// TIA Portal V20 export
FUNCTION_BLOCK "FB2002_Axis_Function"   // FB2, LAD
{ S7_Optimized_Access := 'TRUE' }
// stored: MemoryReserve 100, SetENOAutomatically false
   VAR_INPUT
      Plant_Identifier { ExternalAccessible := 'False'; ExternalVisible := 'False'; ExternalWritable := 'False'} : WString[24];
      Opmode { ExternalAccessible := 'False'; ExternalVisible := 'False'; ExternalWritable := 'False'} : "OPMODE_OUT_UDT";
      TO_Pos_Axis : TO_PositioningAxis;
      Axis_Nr : Int;
      Axis_AbsNum : Int;
      I_SS_bHome : Bool;   // 原点传感器
      I_SS_bFW : Bool := TRUE;   // 前限位
      I_SS_bBW : Bool := TRUE;   // 后限位
      I_CMD_bEnableAxis : Bool;   // 使能
      I_CMD_bResetAxis : Bool;   // 复位
      I_CMD_bjogForward : Bool;   // Taster Aufwärts / 正点
      I_CMD_bjogBackward : Bool;   // Taster Abwärts / 反点
      I_CMD_bmoveVelocity : Bool;   // 速度运行
      I_CMD_bstop : Bool;   // 停止
      I_CMD_bfastStop : Bool;   // 急停
      I_CMD_bHoming : Bool;   // 回零
      I_CMD_bGoToPos : Array[0..15] of Bool;   // Start Aufwärts in Automatik / 16个定位
      I_CMD_iGoToPos : Word;   // 16个定位 Word
      I_CMD_bCallAbsPos : Bool;   // 定位位置切换时，单独的定位按钮
      I_CMD_bRelPos : Bool;   // 相对定位
      I_InLock_bEnableAxis : Bool;   // 使能
      I_InLock_bResetAxis : Bool;   // 复位
      I_InLock_bjogForward : Bool;   // Taster Aufwärts / 正点
      I_InLock_bjogBackward : Bool;   // Taster Abwärts / 反点
      I_InLock_bmoveVelocity : Bool;   // 速度运行
      I_InLock_bstop : Bool;   // 停止
      I_InLock_bfastStop : Bool;   // 急停
      I_InLock_bHoming : Bool;   // 回零
      I_InLock_bGoToPos : Array[0..16] of Bool;   // Start Aufwärts in Automatik / 16个定位
      I_InLock_iGoToPos : Word;   // 16个定位 Word
      I_InLock_bCallAbsPos : Bool;   // 定位位置切换时，单独的定位按钮
      I_InLock_bRelPos : Bool;   // 相对定位
      I_InLock_MyBool : Array[0..5] of Bool;   // 临时变量
      I_CMD_bGoToPos_0 : Bool;   // Start Aufwärts in Automatik / 16个定位自动
      I_InLock_bGoToPos_0 : Bool;   // Start Aufwärts in Automatik / 16个定位条件
      I_CMD_bGoToPos_1 : Bool;   // Start Aufwärts in Automatik / 16个定位自动
      I_InLock_bGoToPos_1 : Bool;   // Start Aufwärts in Automatik / 16个定位条件
      I_CMD_bGoToPos_2 : Bool;   // Start Aufwärts in Automatik / 16个定位自动
      I_InLock_bGoToPos_2 : Bool;   // Start Aufwärts in Automatik / 16个定位条件
      I_CMD_bGoToPos_3 : Bool;   // Start Aufwärts in Automatik / 16个定位自动
      I_InLock_bGoToPos_3 : Bool;   // Start Aufwärts in Automatik / 16个定位条件
      I_CMD_bGoToPos_4 : Bool;   // Start Aufwärts in Automatik / 16个定位自动
      I_InLock_bGoToPos_4 : Bool;   // Start Aufwärts in Automatik / 16个定位条件
      I_CMD_bGoToPos_5 : Bool;   // Start Aufwärts in Automatik / 16个定位自动
      I_InLock_bGoToPos_5 : Bool;   // Start Aufwärts in Automatik / 16个定位条件
      I_CMD_bGoToPos_6 : Bool;   // Start Aufwärts in Automatik / 16个定位自动
      I_InLock_bGoToPos_6 : Bool;   // Start Aufwärts in Automatik / 16个定位条件
      I_CMD_bGoToPos_7 : Bool;   // Start Aufwärts in Automatik / 16个定位自动
      I_InLock_bGoToPos_7 : Bool;   // Start Aufwärts in Automatik / 16个定位条件
      I_CMD_bGoToPos_8 : Bool;   // Start Aufwärts in Automatik / 16个定位自动
      I_InLock_bGoToPos_8 : Bool;   // Start Aufwärts in Automatik / 16个定位条件
   END_VAR
   VAR_OUTPUT
      O_Status_bAxisReady : Bool;   // 轴通讯正常
      O_Status_bAxisEnabled : Bool;   // 轴使能
      O_Status_bjogForward : Bool;   // 轴正点中
      O_Status_bjogBackward : Bool;   // 轴反点中
      O_Status_bHomed : Bool;   // 轴归零完成
      O_Status_bAtHome : Bool;   // 轴在零位
      O_Status_bSstill : Bool;   // 轴静止
      O_Status_bAxisBusy : Bool;   // 轴运行中
      O_Status_bAxisSyned : Bool;   // 同步上
      O_Status_bAxisError : Bool;   // 轴报警
      O_Status_bAtPos : Array[0..15] of Bool;   // Ausgang Aufwärts / 在目标位置上
      O_Status_bPosDone : Array[0..15] of Bool;   // 定位完成
      O_Status_bPosing : Array[0..15] of Bool;   // Ausgang Aufwärts / 定位中
      O_Status_bRelPosDone : Bool;   // 相对定位完成
      O_Status_rActPos : LReal;   // 实际位置
      O_Status_rActSpeed : LReal;   // 实际速度
      O_Status_iAxisFaultNum : UDInt;   // 轴报警代码
      O_Status_iDriveFaultNum : UDInt;   // 驱动报警代码
      O_Status_iFBStatus : Word;   // 运动功能块状态
      O_Status_iMCStatus : Word;   // 运动指令状态
      O_Status_rDriveTorque : LReal;   // 驱动扭矩
      O_Status_rDriveTemp : LReal;   // 驱动温度
      O_Status_rDriveRpm : LReal;   // 驱动转速
      O_Status_AxisName : WString[24] := WSTRING#'No axis';   // Name of axis
      O_Status_mybool : Array[0..5] of Bool;   // 备用
      O_Status_myLreal : Array[0..5] of LReal;   // 备用
   END_VAR
   VAR_IN_OUT
      IF_HMI : "Axis_IF_HMI";
   END_VAR
   VAR
      myFB_Pos16_Ax01 { S7_SetPoint := 'True'} : "FB_Pos16_IO";
      Axis_01 { S7_SetPoint := 'True'} : "FB_Axis";
      i { ExternalAccessible := 'False'; ExternalVisible := 'False'; ExternalWritable := 'False'} : Int;
      j { ExternalAccessible := 'False'; ExternalVisible := 'False'; ExternalWritable := 'False'} : Int;
      HOMIEDONE : Bool;
   END_VAR
BEGIN

REGION Network 1
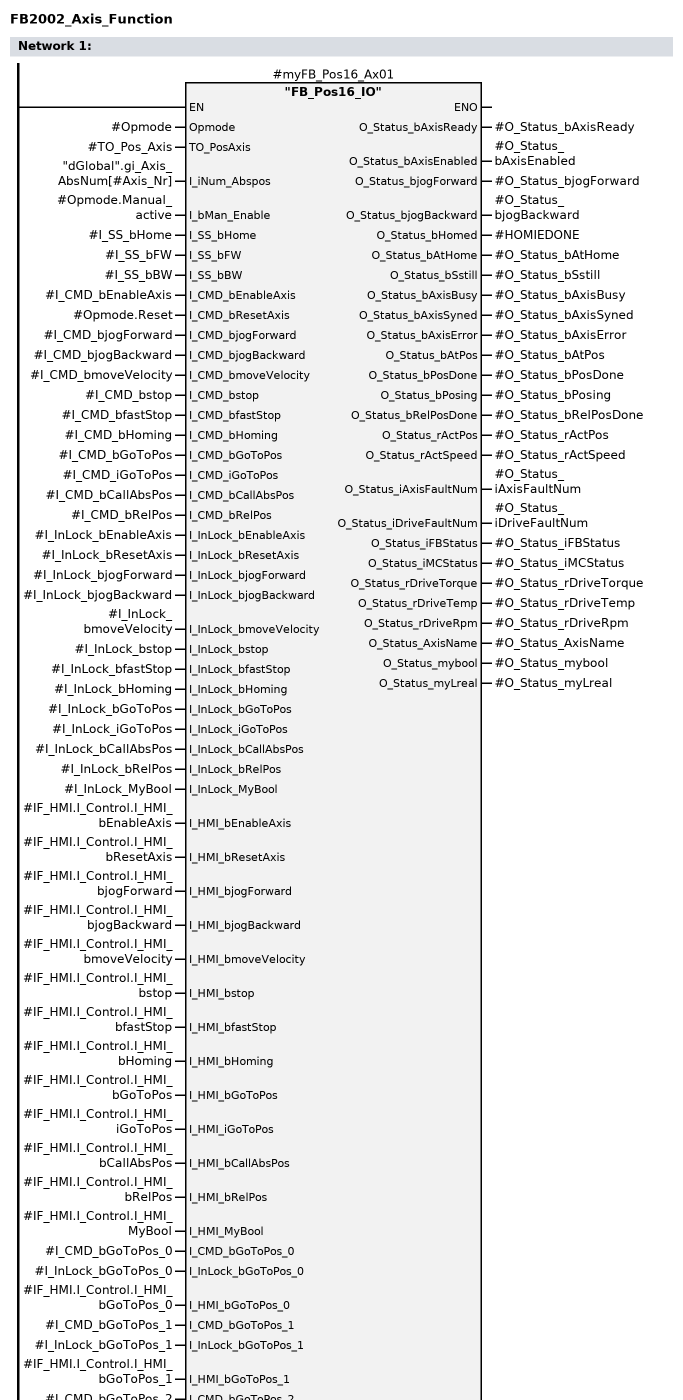
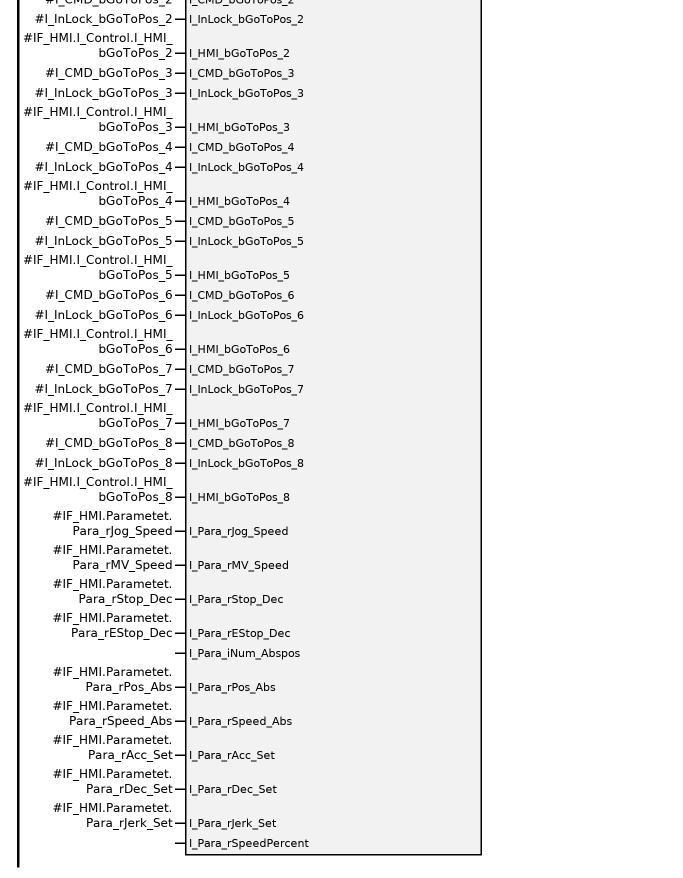
   RUNG wire#powerrail
      #myFB_Pos16_Ax01(Opmode := #Opmode, TO_PosAxis := #TO_Pos_Axis, I_iNum_Abspos := "dGlobal".gi_Axis_AbsNum[#Axis_Nr], I_bMan_Enable := #Opmode.Manual_active, I_SS_bHome := #I_SS_bHome, I_SS_bFW := #I_SS_bFW, I_SS_bBW := #I_SS_bBW, I_CMD_bEnableAxis := #I_CMD_bEnableAxis, I_CMD_bResetAxis := #Opmode.Reset, I_CMD_bjogForward := #I_CMD_bjogForward, I_CMD_bjogBackward := #I_CMD_bjogBackward, I_CMD_bmoveVelocity := #I_CMD_bmoveVelocity, I_CMD_bstop := #I_CMD_bstop, I_CMD_bfastStop := #I_CMD_bfastStop, I_CMD_bHoming := #I_CMD_bHoming, I_CMD_bGoToPos := #I_CMD_bGoToPos, I_CMD_iGoToPos := #I_CMD_iGoToPos, I_CMD_bCallAbsPos := #I_CMD_bCallAbsPos, I_CMD_bRelPos := #I_CMD_bRelPos, I_InLock_bEnableAxis := #I_InLock_bEnableAxis, I_InLock_bResetAxis := #I_InLock_bResetAxis, I_InLock_bjogForward := #I_InLock_bjogForward, I_InLock_bjogBackward := #I_InLock_bjogBackward, I_InLock_bmoveVelocity := #I_InLock_bmoveVelocity, I_InLock_bstop := #I_InLock_bstop, I_InLock_bfastStop := #I_InLock_bfastStop, I_InLock_bHoming := #I_InLock_bHoming, I_InLock_bGoToPos := #I_InLock_bGoToPos, I_InLock_iGoToPos := #I_InLock_iGoToPos, I_InLock_bCallAbsPos := #I_InLock_bCallAbsPos, I_InLock_bRelPos := #I_InLock_bRelPos, I_InLock_MyBool := #I_InLock_MyBool, I_HMI_bEnableAxis := #IF_HMI.I_Control.I_HMI_bEnableAxis, I_HMI_bResetAxis := #IF_HMI.I_Control.I_HMI_bResetAxis, I_HMI_bjogForward := #IF_HMI.I_Control.I_HMI_bjogForward, I_HMI_bjogBackward := #IF_HMI.I_Control.I_HMI_bjogBackward, I_HMI_bmoveVelocity := #IF_HMI.I_Control.I_HMI_bmoveVelocity, I_HMI_bstop := #IF_HMI.I_Control.I_HMI_bstop, I_HMI_bfastStop := #IF_HMI.I_Control.I_HMI_bfastStop, I_HMI_bHoming := #IF_HMI.I_Control.I_HMI_bHoming, I_HMI_bGoToPos := #IF_HMI.I_Control.I_HMI_bGoToPos, I_HMI_iGoToPos := #IF_HMI.I_Control.I_HMI_iGoToPos, I_HMI_bCallAbsPos := #IF_HMI.I_Control.I_HMI_bCallAbsPos, I_HMI_bRelPos := #IF_HMI.I_Control.I_HMI_bRelPos, I_HMI_MyBool := #IF_HMI.I_Control.I_HMI_MyBool, I_CMD_bGoToPos_0 := #I_CMD_bGoToPos_0, I_InLock_bGoToPos_0 := #I_InLock_bGoToPos_0, I_HMI_bGoToPos_0 := #IF_HMI.I_Control.I_HMI_bGoToPos_0, I_CMD_bGoToPos_1 := #I_CMD_bGoToPos_1, I_InLock_bGoToPos_1 := #I_InLock_bGoToPos_1, I_HMI_bGoToPos_1 := #IF_HMI.I_Control.I_HMI_bGoToPos_1, I_CMD_bGoToPos_2 := #I_CMD_bGoToPos_2, I_InLock_bGoToPos_2 := #I_InLock_bGoToPos_2, I_HMI_bGoToPos_2 := #IF_HMI.I_Control.I_HMI_bGoToPos_2, I_CMD_bGoToPos_3 := #I_CMD_bGoToPos_3, I_InLock_bGoToPos_3 := #I_InLock_bGoToPos_3, I_HMI_bGoToPos_3 := #IF_HMI.I_Control.I_HMI_bGoToPos_3, I_CMD_bGoToPos_4 := #I_CMD_bGoToPos_4, I_InLock_bGoToPos_4 := #I_InLock_bGoToPos_4, I_HMI_bGoToPos_4 := #IF_HMI.I_Control.I_HMI_bGoToPos_4, I_CMD_bGoToPos_5 := #I_CMD_bGoToPos_5, I_InLock_bGoToPos_5 := #I_InLock_bGoToPos_5, I_HMI_bGoToPos_5 := #IF_HMI.I_Control.I_HMI_bGoToPos_5, I_CMD_bGoToPos_6 := #I_CMD_bGoToPos_6, I_InLock_bGoToPos_6 := #I_InLock_bGoToPos_6, I_HMI_bGoToPos_6 := #IF_HMI.I_Control.I_HMI_bGoToPos_6, I_CMD_bGoToPos_7 := #I_CMD_bGoToPos_7, I_InLock_bGoToPos_7 := #I_InLock_bGoToPos_7, I_HMI_bGoToPos_7 := #IF_HMI.I_Control.I_HMI_bGoToPos_7, I_CMD_bGoToPos_8 := #I_CMD_bGoToPos_8, I_InLock_bGoToPos_8 := #I_InLock_bGoToPos_8, I_HMI_bGoToPos_8 := #IF_HMI.I_Control.I_HMI_bGoToPos_8, I_Para_rJog_Speed := #IF_HMI.Parametet.Para_rJog_Speed, I_Para_rMV_Speed := #IF_HMI.Parametet.Para_rMV_Speed, I_Para_rStop_Dec := #IF_HMI.Parametet.Para_rStop_Dec, I_Para_rEStop_Dec := #IF_HMI.Parametet.Para_rEStop_Dec, I_Para_iNum_Abspos :=, I_Para_rPos_Abs := #IF_HMI.Parametet.Para_rPos_Abs, I_Para_rSpeed_Abs := #IF_HMI.Parametet.Para_rSpeed_Abs, I_Para_rAcc_Set := #IF_HMI.Parametet.Para_rAcc_Set, I_Para_rDec_Set := #IF_HMI.Parametet.Para_rDec_Set, I_Para_rJerk_Set := #IF_HMI.Parametet.Para_rJerk_Set, I_Para_rSpeedPercent :=, O_Status_bAxisReady => #O_Status_bAxisReady, O_Status_bAxisEnabled => #O_Status_bAxisEnabled, O_Status_bjogForward => #O_Status_bjogForward, O_Status_bjogBackward => #O_Status_bjogBackward, O_Status_bHomed => #HOMIEDONE, O_Status_bAtHome => #O_Status_bAtHome, O_Status_bSstill => #O_Status_bSstill, O_Status_bAxisBusy => #O_Status_bAxisBusy, O_Status_bAxisSyned => #O_Status_bAxisSyned, O_Status_bAxisError => #O_Status_bAxisError, O_Status_bAtPos => #O_Status_bAtPos, O_Status_bPosDone => #O_Status_bPosDone, O_Status_bPosing => #O_Status_bPosing, O_Status_bRelPosDone => #O_Status_bRelPosDone, O_Status_rActPos => #O_Status_rActPos, O_Status_rActSpeed => #O_Status_rActSpeed, O_Status_iAxisFaultNum => #O_Status_iAxisFaultNum, O_Status_iDriveFaultNum => #O_Status_iDriveFaultNum, O_Status_iFBStatus => #O_Status_iFBStatus, O_Status_iMCStatus => #O_Status_iMCStatus, O_Status_rDriveTorque => #O_Status_rDriveTorque, O_Status_rDriveTemp => #O_Status_rDriveTemp, O_Status_rDriveRpm => #O_Status_rDriveRpm, O_Status_AxisName => #O_Status_AxisName, O_Status_mybool => #O_Status_mybool, O_Status_myLreal => #O_Status_myLreal)
   END_RUNG
   // the same network as SCL:
   #myFB_Pos16_Ax01(Opmode := #Opmode,   // "FB_Pos16_IO"
                    TO_PosAxis := #TO_Pos_Axis,
                    I_iNum_Abspos := "dGlobal".gi_Axis_AbsNum[#Axis_Nr],
                    I_bMan_Enable := #Opmode.Manual_active,
                    I_SS_bHome := #I_SS_bHome,
                    I_SS_bFW := #I_SS_bFW,
                    I_SS_bBW := #I_SS_bBW,
                    I_CMD_bEnableAxis := #I_CMD_bEnableAxis,
                    I_CMD_bResetAxis := #Opmode.Reset,
                    I_CMD_bjogForward := #I_CMD_bjogForward,
                    I_CMD_bjogBackward := #I_CMD_bjogBackward,
                    I_CMD_bmoveVelocity := #I_CMD_bmoveVelocity,
                    I_CMD_bstop := #I_CMD_bstop,
                    I_CMD_bfastStop := #I_CMD_bfastStop,
                    I_CMD_bHoming := #I_CMD_bHoming,
                    I_CMD_bGoToPos := #I_CMD_bGoToPos,
                    I_CMD_iGoToPos := #I_CMD_iGoToPos,
                    I_CMD_bCallAbsPos := #I_CMD_bCallAbsPos,
                    I_CMD_bRelPos := #I_CMD_bRelPos,
                    I_InLock_bEnableAxis := #I_InLock_bEnableAxis,
                    I_InLock_bResetAxis := #I_InLock_bResetAxis,
                    I_InLock_bjogForward := #I_InLock_bjogForward,
                    I_InLock_bjogBackward := #I_InLock_bjogBackward,
                    I_InLock_bmoveVelocity := #I_InLock_bmoveVelocity,
                    I_InLock_bstop := #I_InLock_bstop,
                    I_InLock_bfastStop := #I_InLock_bfastStop,
                    I_InLock_bHoming := #I_InLock_bHoming,
                    I_InLock_bGoToPos := #I_InLock_bGoToPos,
                    I_InLock_iGoToPos := #I_InLock_iGoToPos,
                    I_InLock_bCallAbsPos := #I_InLock_bCallAbsPos,
                    I_InLock_bRelPos := #I_InLock_bRelPos,
                    I_InLock_MyBool := #I_InLock_MyBool,
                    I_HMI_bEnableAxis := #IF_HMI.I_Control.I_HMI_bEnableAxis,
                    I_HMI_bResetAxis := #IF_HMI.I_Control.I_HMI_bResetAxis,
                    I_HMI_bjogForward := #IF_HMI.I_Control.I_HMI_bjogForward,
                    I_HMI_bjogBackward := #IF_HMI.I_Control.I_HMI_bjogBackward,
                    I_HMI_bmoveVelocity := #IF_HMI.I_Control.I_HMI_bmoveVelocity,
                    I_HMI_bstop := #IF_HMI.I_Control.I_HMI_bstop,
                    I_HMI_bfastStop := #IF_HMI.I_Control.I_HMI_bfastStop,
                    I_HMI_bHoming := #IF_HMI.I_Control.I_HMI_bHoming,
                    I_HMI_bGoToPos := #IF_HMI.I_Control.I_HMI_bGoToPos,
                    I_HMI_iGoToPos := #IF_HMI.I_Control.I_HMI_iGoToPos,
                    I_HMI_bCallAbsPos := #IF_HMI.I_Control.I_HMI_bCallAbsPos,
                    I_HMI_bRelPos := #IF_HMI.I_Control.I_HMI_bRelPos,
                    I_HMI_MyBool := #IF_HMI.I_Control.I_HMI_MyBool,
                    I_CMD_bGoToPos_0 := #I_CMD_bGoToPos_0,
                    I_InLock_bGoToPos_0 := #I_InLock_bGoToPos_0,
                    I_HMI_bGoToPos_0 := #IF_HMI.I_Control.I_HMI_bGoToPos_0,
                    I_CMD_bGoToPos_1 := #I_CMD_bGoToPos_1,
                    I_InLock_bGoToPos_1 := #I_InLock_bGoToPos_1,
                    I_HMI_bGoToPos_1 := #IF_HMI.I_Control.I_HMI_bGoToPos_1,
                    I_CMD_bGoToPos_2 := #I_CMD_bGoToPos_2,
                    I_InLock_bGoToPos_2 := #I_InLock_bGoToPos_2,
                    I_HMI_bGoToPos_2 := #IF_HMI.I_Control.I_HMI_bGoToPos_2,
                    I_CMD_bGoToPos_3 := #I_CMD_bGoToPos_3,
                    I_InLock_bGoToPos_3 := #I_InLock_bGoToPos_3,
                    I_HMI_bGoToPos_3 := #IF_HMI.I_Control.I_HMI_bGoToPos_3,
                    I_CMD_bGoToPos_4 := #I_CMD_bGoToPos_4,
                    I_InLock_bGoToPos_4 := #I_InLock_bGoToPos_4,
                    I_HMI_bGoToPos_4 := #IF_HMI.I_Control.I_HMI_bGoToPos_4,
                    I_CMD_bGoToPos_5 := #I_CMD_bGoToPos_5,
                    I_InLock_bGoToPos_5 := #I_InLock_bGoToPos_5,
                    I_HMI_bGoToPos_5 := #IF_HMI.I_Control.I_HMI_bGoToPos_5,
                    I_CMD_bGoToPos_6 := #I_CMD_bGoToPos_6,
                    I_InLock_bGoToPos_6 := #I_InLock_bGoToPos_6,
                    I_HMI_bGoToPos_6 := #IF_HMI.I_Control.I_HMI_bGoToPos_6,
                    I_CMD_bGoToPos_7 := #I_CMD_bGoToPos_7,
                    I_InLock_bGoToPos_7 := #I_InLock_bGoToPos_7,
                    I_HMI_bGoToPos_7 := #IF_HMI.I_Control.I_HMI_bGoToPos_7,
                    I_CMD_bGoToPos_8 := #I_CMD_bGoToPos_8,
                    I_InLock_bGoToPos_8 := #I_InLock_bGoToPos_8,
                    I_HMI_bGoToPos_8 := #IF_HMI.I_Control.I_HMI_bGoToPos_8,
                    I_Para_rJog_Speed := #IF_HMI.Parametet.Para_rJog_Speed,
                    I_Para_rMV_Speed := #IF_HMI.Parametet.Para_rMV_Speed,
                    I_Para_rStop_Dec := #IF_HMI.Parametet.Para_rStop_Dec,
                    I_Para_rEStop_Dec := #IF_HMI.Parametet.Para_rEStop_Dec,
                    I_Para_rPos_Abs := #IF_HMI.Parametet.Para_rPos_Abs,
                    I_Para_rSpeed_Abs := #IF_HMI.Parametet.Para_rSpeed_Abs,
                    I_Para_rAcc_Set := #IF_HMI.Parametet.Para_rAcc_Set,
                    I_Para_rDec_Set := #IF_HMI.Parametet.Para_rDec_Set,
                    I_Para_rJerk_Set := #IF_HMI.Parametet.Para_rJerk_Set,
                    O_Status_bAxisReady => #O_Status_bAxisReady,
                    O_Status_bAxisEnabled => #O_Status_bAxisEnabled,
                    O_Status_bjogForward => #O_Status_bjogForward,
                    O_Status_bjogBackward => #O_Status_bjogBackward,
                    O_Status_bHomed => #HOMIEDONE,
                    O_Status_bAtHome => #O_Status_bAtHome,
                    O_Status_bSstill => #O_Status_bSstill,
                    O_Status_bAxisBusy => #O_Status_bAxisBusy,
                    O_Status_bAxisSyned => #O_Status_bAxisSyned,
                    O_Status_bAxisError => #O_Status_bAxisError,
                    O_Status_bAtPos => #O_Status_bAtPos,
                    O_Status_bPosDone => #O_Status_bPosDone,
                    O_Status_bPosing => #O_Status_bPosing,
                    O_Status_bRelPosDone => #O_Status_bRelPosDone,
                    O_Status_rActPos => #O_Status_rActPos,
                    O_Status_rActSpeed => #O_Status_rActSpeed,
                    O_Status_iAxisFaultNum => #O_Status_iAxisFaultNum,
                    O_Status_iDriveFaultNum => #O_Status_iDriveFaultNum,
                    O_Status_iFBStatus => #O_Status_iFBStatus,
                    O_Status_iMCStatus => #O_Status_iMCStatus,
                    O_Status_rDriveTorque => #O_Status_rDriveTorque,
                    O_Status_rDriveTemp => #O_Status_rDriveTemp,
                    O_Status_rDriveRpm => #O_Status_rDriveRpm,
                    O_Status_AxisName => #O_Status_AxisName,
                    O_Status_mybool => #O_Status_mybool,
                    O_Status_myLreal => #O_Status_myLreal);
END_REGION

REGION Network 2 (SCL)
   IF #HOMIEDONE THEN
       #O_Status_bHomed := 1;
   END_IF;
   IF #O_Status_rActSpeed>0.5 THEN
           #O_Status_bHomed := 0;
   END_IF;
END_REGION

REGION Network 4 (SCL)


       "dGlobal".gi_Axis_AbsNum[#Axis_Nr] := #Axis_AbsNum;
END_REGION

REGION Network 6 (SCL)

       "dStruct_Axis".gs_Axis[#Axis_Nr].I_CMD.bResetAxis := #Opmode.Reset;
       "dStruct_Axis".gs_Axis[#Axis_Nr].I_InLock.bjogForward := "dStruct_Axis".gs_Axis[#Axis_Nr].O_Status.bAxisEnabled;
       "dStruct_Axis".gs_Axis[#Axis_Nr].I_InLock.bjogBackward := "dStruct_Axis".gs_Axis[#Axis_Nr].O_Status.bAxisEnabled;
       "dStruct_Axis".gs_Axis[#Axis_Nr].I_InLock.bHoming := true;
       FOR #j := 0 TO 16 DO
           "dStruct_Axis".gs_Axis[#Axis_Nr].I_InLock.bGoToPos[#j] := true;
       END_FOR;


       IF "dGlobal".Old_Pos_Select <> "dGlobal".gbo_Pos_Select THEN//刚切换
           "dStruct_Axis".gs_Axis[0].I_Para.rPos_Abs[0] := "dStruct_Axis".gs_Axis["dGlobal".gbo_Axis_Select].I_Para.rPos_Abs["dGlobal".gbo_Pos_Select];
           "dStruct_Axis".gs_Axis[0].I_Para.rSpeed_Abs[0] := "dStruct_Axis".gs_Axis["dGlobal".gbo_Axis_Select].I_Para.rSpeed_Abs["dGlobal".gbo_Pos_Select];

           "dGlobal".Old_Pos_Select := "dGlobal".gbo_Pos_Select;
       ELSE
           "dStruct_Axis".gs_Axis["dGlobal".gbo_Axis_Select].I_Para.rPos_Abs["dGlobal".gbo_Pos_Select] := "dStruct_Axis".gs_Axis[0].I_Para.rPos_Abs[0];
           "dStruct_Axis".gs_Axis["dGlobal".gbo_Axis_Select].I_Para.rSpeed_Abs["dGlobal".gbo_Pos_Select] := "dStruct_Axis".gs_Axis[0].I_Para.rSpeed_Abs[0];
       END_IF;
END_REGION

REGION Network 7 (SCL)
   #IF_HMI.Show_Sensor.I_SS_bHome := #I_SS_bHome;
   #IF_HMI.Show_Sensor.I_SS_bFW := #I_SS_bFW;
   #IF_HMI.Show_Sensor.I_SS_bBW := #I_SS_bBW;
   #IF_HMI.O_Status.O_Status_bAxisReady := #O_Status_bAxisReady;
   #IF_HMI.O_Status.O_Status_bAxisEnabled := #O_Status_bAxisEnabled;
   #IF_HMI.O_Status.O_Status_bjogForward := #O_Status_bjogForward;
   #IF_HMI.O_Status.O_Status_bjogBackward := #O_Status_bjogBackward;
   #IF_HMI.O_Status.O_Status_bHomed := #O_Status_bHomed;
   #IF_HMI.O_Status.O_Status_bAtHome := #O_Status_bAtHome;
   #IF_HMI.O_Status.O_Status_bSstill := #O_Status_bSstill;
   #IF_HMI.O_Status.O_Status_bAxisBusy := #O_Status_bAxisBusy;
   #IF_HMI.O_Status.O_Status_bAxisSyned := #O_Status_bAxisSyned;
   #IF_HMI.O_Status.O_Status_bAxisError := #O_Status_bAxisError;
   #IF_HMI.O_Status.O_Status_bAtPos := #O_Status_bAtPos;
   #IF_HMI.O_Status.O_Status_bPosDone := #O_Status_bPosDone;
   #IF_HMI.O_Status.O_Status_bPosing := #O_Status_bPosing;
   #IF_HMI.O_Status.O_Status_bRelPosDone := #O_Status_bRelPosDone;
   #IF_HMI.O_Status.O_Status_rActPos := #O_Status_rActPos;
   #IF_HMI.O_Status.O_Status_rActSpeed := #O_Status_rActSpeed;
   #IF_HMI.O_Status.O_Status_iAxisFaultNum := #O_Status_iAxisFaultNum;
   #IF_HMI.O_Status.O_Status_iDriveFaultNum := #O_Status_iDriveFaultNum;
   #IF_HMI.O_Status.O_Status_iFBStatus := #O_Status_iFBStatus;
   #IF_HMI.O_Status.O_Status_iMCStatus := #O_Status_iMCStatus;
   #IF_HMI.O_Status.O_Status_rDriveTorque := #O_Status_rDriveTorque;
   #IF_HMI.O_Status.O_Status_rDriveTemp := #O_Status_rDriveTemp;
   #IF_HMI.O_Status.O_Status_rDriveRpm := #O_Status_rDriveRpm;
   #IF_HMI.O_Status.O_Status_AxisName := #O_Status_AxisName;
   #IF_HMI.O_Status.O_Status_mybool := #O_Status_mybool;
   #IF_HMI.O_Status.O_Status_myLreal := #O_Status_myLreal;
   #IF_HMI.Plant_Identifier := #Plant_Identifier;
END_REGION

REGION Network 8 (SCL)
   "dGlobal".gi_Axis_AbsNum[0] := "dGlobal".gi_Axis_AbsNum["dGlobal".gbo_Axis_Select];
END_REGION
END_FUNCTION_BLOCK
